// TIA Portal project "limit switch" (V16)

(* hardware
DEVICE "S7-1200 station_1"  S7-1200 Station
   slot 0: "Rack_0"  S7-1200 Rack  Rack  V1.0
   slot 1: "PLC_1"  CPU 1212C AC/DC/Rly  6ES7 212-1BE40-0XB0  V4.0
*)

// ===== PLC "PLC_1"  CPU 1212C AC/DC/Rly =====

VAR_GLOBAL   // PLC tag table "Default tag table"
   "K1" AT %Q0.0 : Bool;
   "k2" AT %Q0.1 : Bool;
   "X" AT %M0.2 : Bool;
   "K3" AT %Q0.2 : Bool;
   "start1" AT %I0.2 : Bool;
   "Tag_2" AT %M0.1 : Bool;
   "L2 Run" AT %M0.3 : Bool;
   "Tag_4" AT %M0.4 : Bool;
   "Tag_5" AT %M1.1 : Bool;
   "Tag_6" AT %M1.0 : Bool;
   "stop condition" AT %M0.5 : Bool;
   "STOP" AT %I0.3 : Bool;
   "L2" AT %I0.5 : Bool;
   "L3" AT %I0.6 : Bool;
   "L1" AT %I0.4 : Bool;
   "Tag_1" AT %I0.1 : Bool;
END_VAR

ORGANIZATION_BLOCK "Main"   // OB1, LAD, ProgramCycle
TITLE = "Main Program Sweep (Cycle)"
{ S7_Optimized_Access := 'TRUE' }
VERSION : 0.1
   VAR_INPUT
      Initial_Call : Bool;   // Initial call of this OB
      Remanence : Bool;   // =True, if remanent data are available
   END_VAR
BEGIN

REGION Network 1: start
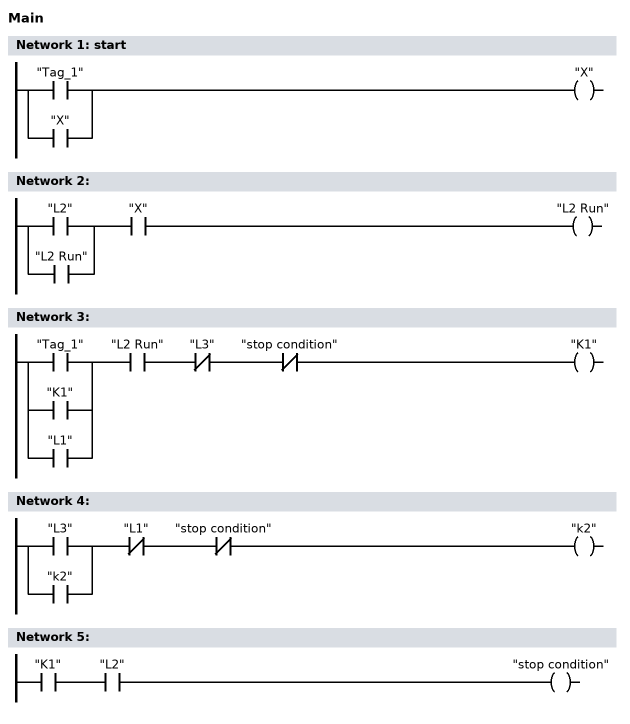
   RUNG wire#powerrail
      Contact( "Tag_1" )
      wire#w1
      Coil( "X" )
   END_RUNG
   RUNG wire#powerrail
      Contact( "X" )
   END_RUNG wire#w1
   // the same network as SCL:
   "X" := "Tag_1" OR "X";
END_REGION

REGION Network 2
   RUNG wire#powerrail
      Contact( "L2" )
      wire#w1
      Contact( "X" )
      Coil( "L2 Run" )
   END_RUNG
   RUNG wire#powerrail
      Contact( "L2 Run" )
   END_RUNG wire#w1
   // the same network as SCL:
   "L2 Run" := ("L2" OR "L2 Run") AND "X";
END_REGION

REGION Network 3
   RUNG wire#powerrail
      Contact( "Tag_1" )
      wire#w1
      Contact( "L2 Run" )
      I_Contact( "L3" )
      I_Contact( "stop condition" )
      Coil( "K1" )
   END_RUNG
   RUNG wire#powerrail
      Contact( "K1" )
   END_RUNG wire#w1
   RUNG wire#powerrail
      Contact( "L1" )
   END_RUNG wire#w1
   // the same network as SCL:
   "K1" := ("Tag_1" OR "K1" OR "L1") AND "L2 Run" AND NOT "L3" AND NOT "stop condition";
END_REGION

REGION Network 4
   RUNG wire#powerrail
      Contact( "L3" )
      wire#w1
      I_Contact( "L1" )
      I_Contact( "stop condition" )
      Coil( "k2" )
   END_RUNG
   RUNG wire#powerrail
      Contact( "k2" )
   END_RUNG wire#w1
   // the same network as SCL:
   "k2" := ("L3" OR "k2") AND NOT "L1" AND NOT "stop condition";
END_REGION

REGION Network 5
   RUNG wire#powerrail
      Contact( "K1" )
      Contact( "L2" )
      Coil( "stop condition" )
   END_RUNG
   // the same network as SCL:
   "stop condition" := "K1" AND "L2";
END_REGION
END_ORGANIZATION_BLOCK